// TIA Portal V15.1 export
// export: Created 2020-06-12T07:35:46.5380859Z, ExportSetting None, DisplayName Totally Integrated Automation Portal, DisplayVersion V15.1, DisplayName TIA Portal Openness, DisplayVersion V15.1, DisplayName STEP 7 Professional, DisplayVersion V15.1, DisplayName STEP 7 Safety, DisplayVersion V15.1, DisplayName WinCC Advanced, DisplayVersion V15.1
FUNCTION "ELC_call" : Void   // FC86, FBD
TITLE = Electrode carriage call
{ S7_Optimized_Access := 'TRUE' }
// stored: SetENOAutomatically False
BEGIN

REGION Network 1: Movement
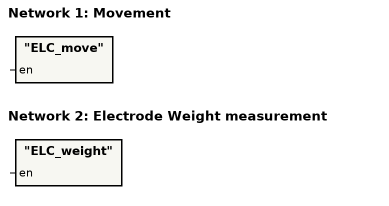
   "ELC_move"();
END_REGION

REGION Network 2: Electrode Weight measurement
   "ELC_weight"();
END_REGION
END_FUNCTION
